// TIA Portal V21 export
FUNCTION "Motore_PompaPistoni" : Void   // FC132, LAD
{ S7_Optimized_Access := 'TRUE' }
// stored: SetENOAutomatically false
   VAR_TEMP
      AutoPos : Bool;
      AutoNeg : Bool;
      VolumeTeorico : Real;
      DeltaVolume : Real;
      MassimoDeltaScostamento : Real;
   END_VAR
BEGIN

REGION Network 1: Comando positivo in automatico
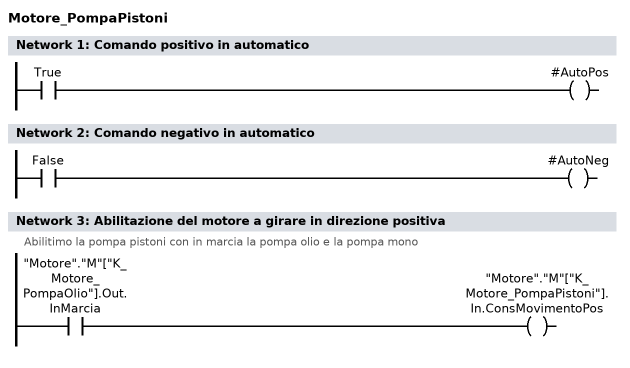
   RUNG wire#powerrail
      Contact( True )
      Coil( #AutoPos )
   END_RUNG
   // the same network as SCL:
   #AutoPos := True;
END_REGION

REGION Network 2: Comando negativo in automatico
   RUNG wire#powerrail
      Contact( False )
      Coil( #AutoNeg )
   END_RUNG
   // the same network as SCL:
   #AutoNeg := False;
END_REGION

REGION Network 3: Abilitazione del motore a girare in direzione positiva
   // Abilitimo la pompa pistoni con in marcia la pompa olio e la pompa mono
   RUNG wire#powerrail
      Contact( "Motore"."M"["K_Motore_PompaOlio"].Out.InMarcia )
      Coil( "Motore"."M"["K_Motore_PompaPistoni"].In.ConsMovimentoPos )
   END_RUNG
   // the same network as SCL:
   "Motore"."M"["K_Motore_PompaPistoni"].In.ConsMovimentoPos := "Motore"."M"["K_Motore_PompaOlio"].Out.InMarcia;
END_REGION

REGION Network 4 (SCL)
   REGION PompaPistoni
       REGION Ingressi
           "Motore".M[K_Motore_PompaPistoni].In.FbDigitali.FaultInverter := NOT "PompaPistoni_Ready";
           "Motore".M[K_Motore_PompaPistoni].In.FbDigitali.FeedbackMarcia := "PompaPistoni_Marcia";
           "Motore".M[K_Motore_PompaPistoni].Prm.Generali.K_Analogica := "K_Analogica_PortataIngressoProdotto";
           // "Motore".M["K_Motore_PompaPistoni"].In.CmdPosRich := #AutoPos;
           // "Motore".M["K_Motore_PompaPistoni"].In.CmdPosRich := #AutoNeg;
       END_REGION ;
       REGION Gestione
           "GestMotore"(K_Motore := "K_Motore_PompaPistoni",
                        K_TipoMotore := "K_TipoMotore_InverterKEB",
                        K_Zona := "K_Zona_Sterilizzatore");

           "GestMotore_Servoventola"(K_Motore := "K_Motore_PompaPistoni",
                                     TermicoScattato := NOT "PompaPistoni_Ventola_TermicoOk",
                                     ComandoMarcia => "PompaPistoni_Servoventola_ComandoMarcia");
       END_REGION ;
       REGION Uscite
           "PompaPistoni_ComandoMarcia" := "Motore".M[K_Motore_PompaPistoni].Out.CmdPosMotore;
           "PompaPistoni_ResetInverter" := "Motore".M[K_Motore_PompaPistoni].In.Reset;
           "PompaPistoni_Velocità" := DINT_TO_WORD("Motore".M[K_Motore_PompaPistoni].Out.Paw);
       END_REGION ;
   END_REGION ;
END_REGION

REGION Network 5 (SCL): Gestione allarme inseguimento
   REGION Gestione dell'allarme inseguimento
       REGION Calcoli
           #VolumeTeorico := "Motore".M[K_Motore_PompaPistoni].Dati.FrequenzaRichiesta * 153.85 + 57.692;                        //Volume teorico calcolato sulla base della frequenza attuale
           #DeltaVolume := ABS(#VolumeTeorico - "Motore".M[K_Motore_PompaPistoni].Dati.Feedback_Speed);                          //Differenza tra il valore teroico e quella reale 
           #MassimoDeltaScostamento := 200.0;                                                                                      //Massimo delta di scostamento accettabile prima di dare allarme
       END_REGION ;
       REGION Timer                                                    
           "T_ON"(I_CicloCPU := "CicloScansioneCPU_I".O_rCicloCpu,                                                                 //Ritardo
                  I_StartConteggio := "Motore".M[K_Motore_PompaPistoni].Out.CmdPosMotore,                                        //alla partenza del motore
                  IO_DatiTimer := "Pompapistoni_Timer".RitardoPartenza);                                                           //Per ritardardare l'allarme
           "T_ON"(I_CicloCPU := "CicloScansioneCPU_I".O_rCicloCpu,                                                                 //Ritardo
                  I_StartConteggio := #DeltaVolume > #MassimoDeltaScostamento AND "Pompapistoni_Timer".RitardoPartenza.O,          //Di scostamento
                  IO_DatiTimer := "Pompapistoni_Timer".RitardoInAllarme);                                                          //Dal massimo delta possibile
       END_REGION ;
       REGION Set allarme
           "Motore".M[K_Motore_PompaPistoni].Allarmi.A[KAllMot_FollowingError].Stato := "Pompapistoni_Timer".RitardoInAllarme.O;
       END_REGION ;
   END_REGION ;
END_REGION
END_FUNCTION
